SUBAPPLICATION Uebung_080c_AUI (* Beispiel für E_CTU mit AX_T_FF und AX_PERMIT (Event-Halbierung) und Terminal-Ausgabe *)
  (* Standard: 61499-2; Description: Copyright (c) 2023 Meisterschulen am Ostbahnhof This program and the accompanying materials are made available under the terms of the Eclipse Public License 2.0 which is available at https://www.eclipse.org/legal/epl-2.0/ SPDX-License-Identifier: EPL-2.0 *)
  (* Version 1.1, 2026-04-21, Franz Höpfinger, Meisterschulen am Ostbahnhof, Added terminal output for counter value *)
  PACKAGE Uebungen;
  IMPORT Uebungen::const::UT::DefaultPool::OutputNumber_N1;
  IMPORT logiBUS::io::DI::logiBUS_DI::Input_I1;
  IMPORT logiBUS::io::DI::logiBUS_DI::Input_I2;
  IMPORT logiBUS::io::DI::logiBUS_DI_Events::BUTTON_SINGLE_CLICK;
  IMPORT logiBUS::io::DQ::logiBUS_DO::Output_Q1;
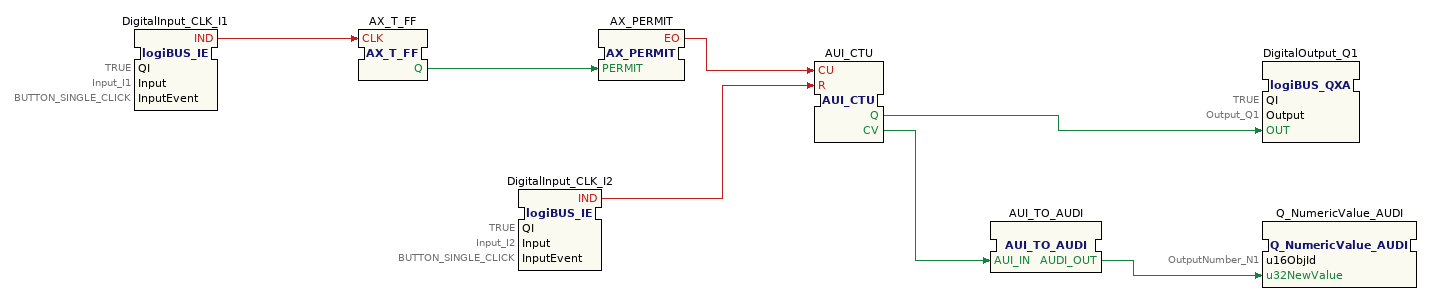
  FBS
    DigitalOutput_Q1 : logiBUS::io::DQ::logiBUS_QXA(QI := TRUE, Output := Output_Q1);
    DigitalInput_CLK_I1 : logiBUS::io::DI::logiBUS_IE(QI := TRUE, Input := Input_I1, InputEvent := BUTTON_SINGLE_CLICK);
    AUI_CTU : adapter::events::unidirectional::AUI_CTU;
    DigitalInput_CLK_I2 : logiBUS::io::DI::logiBUS_IE(QI := TRUE, Input := Input_I2, InputEvent := BUTTON_SINGLE_CLICK);
    AX_PERMIT : adapter::events::unidirectional::AX_PERMIT;
    AX_T_FF : adapter::events::unidirectional::AX_T_FF;
    AUI_TO_AUDI : adapter::conversion::unidirectional::AUI_TO_AUDI;
    Q_NumericValue_AUDI : isobus::UT::Q::Q_NumericValue_AUDI(u16ObjId := OutputNumber_N1);
  END_FBS
  EVENT_CONNECTIONS
    DigitalInput_CLK_I1.IND TO AX_T_FF.CLK;
    AX_PERMIT.EO TO AUI_CTU.CU;
    DigitalInput_CLK_I2.IND TO AUI_CTU.R;
  END_CONNECTIONS
  ADAPTER_CONNECTIONS
    AX_T_FF.Q TO AX_PERMIT.PERMIT;
    AUI_CTU.Q TO DigitalOutput_Q1.OUT;
    AUI_CTU.CV TO AUI_TO_AUDI.AUI_IN;
    AUI_TO_AUDI.AUDI_OUT TO Q_NumericValue_AUDI.u32NewValue;
  END_CONNECTIONS
END_SUBAPPLICATION
